{attribute 'linkalways'} 
{attribute 'no_explicit_call' := 'This FB is a CLASS and must be accessed using methods or properties'}
{attribute 'enable_dynamic_creation'}
FUNCTION_BLOCK FINAL LE_DINT EXTENDS Node
VAR
	in1 : _DINT(0);
	in2 : _DINT(0);
	out : _BOOL(FALSE);
END_VAR

METHOD PUBLIC Clone : I_Node
VAR
	pNode : POINTER TO LE_DINT;
END_VAR
pNode := __NEW(LE_DINT);
Clone := pNode^;
END_METHOD

METHOD FB_init : BOOL
VAR_INPUT
	bInitRetains : BOOL; // if TRUE, the retain variables are initialized (warm start / cold start)
	bInCopyCode : BOOL;  // if TRUE, the instance afterwards gets moved into the copy code (online change)
END_VAR
AddInput('in1',THIS^.in1);
AddInput('in2',THIS^.in2);
AddOutput('out', THIS^.out);
END_METHOD

METHOD PROTECTED OnExecute
VAR
END_VAR
out.Value := in1.Value <= in2.Value;
END_METHOD

END_FUNCTION_BLOCK

(* stored: Version 1.1.0.1, ProductVersion 3.1.4024.15
   POU LE_DINT: Id {b9e3f839-d3a6-49fa-ba32-bb32c29a2995}, SpecialFunc None
   Folder Constructor: Id {dac1a3e3-382a-40f1-859e-69493eebe9e6}
   Method Clone: Id {253e147e-934a-47a6-8395-0297e4ca39ff}
   Method FB_init: Id {f51477af-f6fe-435b-baa5-e883eaac0c18}
   Method OnExecute: Id {fd91e075-ad10-4fc2-8d90-c97ec72df1f0} *)
